// Mitsubishi GX Works2 project: USANDO FUCTION   PLC: Q03UDV

// task Task_01 (event TRUE, interval 0, priority 31): POU_01

PROGRAM POU_01
VAR
  CTD_1 : CTD;
END_VAR
(* structured ladder/FBD written out as ST: instructions are called as NAME(EN, inputs, outputs); _pN, _eN, _tN stand for wires *)
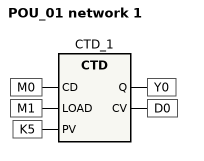
(* network 1 *)
CTD_1(CD := M0, LOAD := M1, PV := K5, Q => Y0, CV => D0);
END_PROGRAM
